FUNCTION_BLOCK SPLIT_SIGNED_REAL (* Teilt einen REAL-Wert in 2 einseitige Betragswerte auf: NEG_MAG = MAX(0,-Y), POS_MAG = MAX(0,Y). Feuert CNF bei jedem REQ, unabhaengig von Wertaenderung - Event-Deduplizierung erfolgt aussen im Adapter-Wrapper AR_SPLIT_SIGNED ueber je einen E_D_FF_ANY pro Seite. *)
  (* Standard: 61499-2 *)
  (* Version 1.0, 2026-09-11, Franz Höpfinger, Einfacher Value/Event-Baustein ohne Event-Dedup - wird vom Adapter-Wrapper AR_SPLIT_SIGNED mit je einem E_D_FF_ANY pro Seite dedupliziert *)
  PACKAGE adapter::Engineering::splitting::signed;
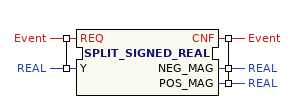
  EVENT_INPUT
    REQ WITH Y; (* Neuer Y-Wert liegt an *)
  END_EVENT
  EVENT_OUTPUT
    CNF WITH NEG_MAG, POS_MAG; (* NEG_MAG/POS_MAG berechnet *)
  END_EVENT
  VAR_INPUT
    Y : REAL; (* Eingangswert *)
  END_VAR
  VAR_OUTPUT
    NEG_MAG : REAL; (* MAX(0, -Y) *)
    POS_MAG : REAL; (* MAX(0, Y) *)
  END_VAR
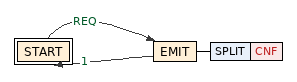
  EC_STATES
    START; (* Initial State *)
    EMIT : SPLIT -> CNF;
  END_STATES
  EC_TRANSITIONS
    START TO EMIT := REQ;
    EMIT TO START := 1;
  END_TRANSITIONS
  ALGORITHM SPLIT IN ST:
NEG_MAG := MAX(REAL#0.0,-Y);
POS_MAG := MAX(REAL#0.0,Y);
  END_ALGORITHM
END_FUNCTION_BLOCK
